{attribute 'Tc2GvlVarNames'}
VAR_GLOBAL
	TCP_SERVER_RESET : BYTE; (* nur für TwinCAT notwendig ! *)
	LOG_CL : LOG_CONTROL;
END_VAR

(* stored: Version 1.1.0.1, ProductVersion 3.1.4022.7
   GVL Globale_Variablen_1: Id {bd319891-649f-44f9-aa4e-1cd61161dc03} *)
